(* IEC 61131-3 sources: CodigoPPC/FB Com, 4 files *)

(* ---- FB_CheckInversores.st ---- *)
(* ═══════════════════════════════════════════════════════════════════════
   FB_CheckInversores (NOVA VERSÃO — ModbusFB programático)
   ═══════════════════════════════════════════════════════════════════════
   INTERFACE EXTERNA PRESERVADA — FB_Startup não precisa mudar:
     - Mesmos VAR_INPUT: xEnable, tTxTimeout, tGlobalTimeout
     - Mesmos VAR_OUTPUT: xDone, xFailed, uRespondedTotal, uConfiguredTotal,
       uLastFailIdx, uLastFailCOM

   MUDANÇA INTERNA:
     - Removido: FB_ModBus (antigo) com triggers e ModbusSlaveComPort
     - Adicionado: ClientRequestReadHoldingRegisters via referência a ClientSerial
     - Lê slave IDs da configuração (GVL_Comm) ao invés de ponteiros do Device Tree

   A varredura permanece sequencial: 1 transação por ciclo de scan,
   COM1 primeiro, depois COM2.
   ═══════════════════════════════════════════════════════════════════════ *)
FUNCTION_BLOCK FB_CheckInversores

VAR_INPUT
    xEnable         : BOOL;
    tTxTimeout      : TIME := T#500MS;
    tGlobalTimeout  : TIME := T#60S;
END_VAR

VAR_IN_OUT
    rClientCOM1     : ModbusFB.ClientSerial;    // Referência ao client COM1
    rClientCOM2     : ModbusFB.ClientSerial;    // Referência ao client COM2
    // Arrays de slave IDs por porta COM
    auiSlaveIdsCOM1 : ARRAY[1..15] OF UINT;    // Slave IDs inversores COM1
    auiSlaveIdsCOM2 : ARRAY[1..15] OF UINT;    // Slave IDs inversores COM2
END_VAR

VAR_OUTPUT
    xDone           : BOOL;
    xFailed         : BOOL;
    uRespondedTotal : UINT;
    uConfiguredTotal: UINT;
    uLastFailIdx    : UINT;
    uLastFailCOM    : UINT;
END_VAR

VAR
    _fbRead         : ModbusFB.ClientRequestReadHoldingRegisters;
    _awBuf          : ARRAY[0..1] OF WORD;      // buffer mínimo para leitura de teste

    uCheckIdx       : UINT := 1;
    uCheckCOM       : UINT := 1;                // 1=COM1, 2=COM2, 3=avaliação
    uRespondedCOM1  : UINT := 0;
    uRespondedCOM2  : UINT := 0;
    bInitDone       : BOOL := FALSE;
    bReqInitDone    : BOOL := FALSE;
    TonGlobal       : TON;
    CheckThreshold  : REAL := 1.0;

    _state          : (CS_IDLE, CS_SENDING, CS_WAITING) := CS_IDLE;
    _uiRegAddr      : UINT := 0;               // Endereço de teste (reg 0 — qualquer holding register)
END_VAR

    // ── Reset quando desabilitado ────────────────────────────────────
    IF NOT xEnable THEN
        xDone            := FALSE;
        xFailed          := FALSE;
        uRespondedCOM1   := 0;
        uRespondedCOM2   := 0;
        uRespondedTotal  := 0;
        uConfiguredTotal := 0;
        uLastFailIdx     := 0;
        uLastFailCOM     := 0;
        uCheckIdx        := 1;
        uCheckCOM        := 1;
        bInitDone        := FALSE;
        bReqInitDone     := FALSE;
        _state           := CS_IDLE;
        TonGlobal(IN := FALSE);
        RETURN;
    END_IF

    // Se já terminou, mantém resultado
    IF xDone OR xFailed THEN
        RETURN;
    END_IF

    // Inicialização
    IF NOT bInitDone THEN
        uConfiguredTotal := GVL_Main.NInversoresCOM01 + GVL_Main.NInversoresCOM02;
        bInitDone := TRUE;
    END_IF

    // Inicialização do request (uma vez)
    IF NOT bReqInitDone THEN
        _fbRead(
            rClient     := rClientCOM1,
            udiTimeout  := TIME_TO_UDINT(tTxTimeout) * 1000,
            uiMaxRetries := 0   // Sem retry no check — queremos saber rápido
        );
        bReqInitDone := TRUE;
    END_IF

    // Chamar request a cada ciclo (obrigatório)
    IF uCheckCOM <= 1 THEN
        _fbRead(rClient := rClientCOM1);
    ELSE
        _fbRead(rClient := rClientCOM2);
    END_IF

    // Timeout global
    TonGlobal(IN := TRUE, PT := tGlobalTimeout);
    IF TonGlobal.Q THEN
        TonGlobal(IN := FALSE);
        uRespondedTotal := uRespondedCOM1 + uRespondedCOM2;
        xFailed := TRUE;
        RETURN;
    END_IF

    // ── Varredura COM1 ──────────────────────────────────────────────
    IF uCheckCOM = 1 THEN
        IF uCheckIdx <= GVL_Main.NInversoresCOM01 THEN

            CASE _state OF
                CS_IDLE:
                    // Disparar leitura de 1 registro do inversor atual
                    _fbRead(
                        rClient     := rClientCOM1,
                        xExecute    := TRUE,
                        uiUnitId    := auiSlaveIdsCOM1[uCheckIdx],
                        uiStartItem := _uiRegAddr,
                        uiQuantity  := 1,
                        pData       := ADR(_awBuf[0])
                    );
                    _state := CS_WAITING;

                CS_WAITING:
                    IF _fbRead.xDone THEN
                        _fbRead.xExecute := FALSE;
                        uRespondedCOM1 := uRespondedCOM1 + 1;
                        GVL_Comm.abInvOnline_COM1[uCheckIdx] := TRUE;
                        uCheckIdx := uCheckIdx + 1;
                        _state := CS_IDLE;

                    ELSIF _fbRead.xError THEN
                        _fbRead.xExecute := FALSE;
                        uLastFailIdx := uCheckIdx;
                        uLastFailCOM := 1;
                        GVL_Comm.abInvOnline_COM1[uCheckIdx] := FALSE;
                        uCheckIdx := uCheckIdx + 1;
                        _state := CS_IDLE;
                    END_IF
                    // BUSY: aguarda
            END_CASE

        ELSE
            // COM1 concluída — avançar para COM2
            uCheckIdx := 1;
            uCheckCOM := 2;
            _state := CS_IDLE;
        END_IF

    // ── Varredura COM2 ──────────────────────────────────────────────
    ELSIF uCheckCOM = 2 THEN
        IF GVL_Main.NInversoresCOM02 = 0 THEN
            uCheckCOM := 3;

        ELSIF uCheckIdx <= GVL_Main.NInversoresCOM02 THEN

            CASE _state OF
                CS_IDLE:
                    _fbRead(
                        rClient     := rClientCOM2,
                        xExecute    := TRUE,
                        uiUnitId    := auiSlaveIdsCOM2[uCheckIdx],
                        uiStartItem := _uiRegAddr,
                        uiQuantity  := 1,
                        pData       := ADR(_awBuf[0])
                    );
                    _state := CS_WAITING;

                CS_WAITING:
                    IF _fbRead.xDone THEN
                        _fbRead.xExecute := FALSE;
                        uRespondedCOM2 := uRespondedCOM2 + 1;
                        GVL_Comm.abInvOnline_COM2[uCheckIdx] := TRUE;
                        uCheckIdx := uCheckIdx + 1;
                        _state := CS_IDLE;

                    ELSIF _fbRead.xError THEN
                        _fbRead.xExecute := FALSE;
                        uLastFailIdx := uCheckIdx;
                        uLastFailCOM := 2;
                        GVL_Comm.abInvOnline_COM2[uCheckIdx] := FALSE;
                        uCheckIdx := uCheckIdx + 1;
                        _state := CS_IDLE;
                    END_IF
            END_CASE

        ELSE
            uCheckCOM := 3;
        END_IF

    // ── Avaliação final ─────────────────────────────────────────────
    ELSIF uCheckCOM = 3 THEN
        TonGlobal(IN := FALSE);
        uRespondedTotal := uRespondedCOM1 + uRespondedCOM2;

        IF uConfiguredTotal = 0 THEN
            xFailed := TRUE;
            RETURN;
        END_IF

        IF (TO_REAL(uRespondedTotal) / TO_REAL(uConfiguredTotal)) >= CheckThreshold THEN
            xDone := TRUE;
        ELSE
            xFailed := TRUE;
        END_IF

        GVL_Comm.uiInvOnlineCount_COM1 := uRespondedCOM1;
        GVL_Comm.uiInvOnlineCount_COM2 := uRespondedCOM2;
    END_IF
END_FUNCTION_BLOCK

(* ---- FB_ModBus.st ---- *)
(* ═══════════════════════════════════════════════════════════════════════
   FB_ModBus (NOVA VERSÃO — ModbusFB programático)
   ═══════════════════════════════════════════════════════════════════════
   Substitui o FB_ModBus anterior que usava triggers booleanos e
   ModbusSlaveComPort do Device Tree.

   Esta versão encapsula um ClientRequestReadHoldingRegisters do ModbusFB,
   mantendo a MESMA INTERFACE EXTERNA (E_ModbusResult) para que:
     - FB_WriteCom, FB_CheckInversores e FB_Startup não precisem mudar
       sua lógica interna de tratamento de resultado.

   MUDANÇA PRINCIPAL:
     Antes: trigInv (BOOL) + pSlave (ModbusSlaveComPort) → rising edge no driver
     Agora: xExecute + rClient (ClientSerial) + uiUnitId + uiStartItem + pData

   CONTRATO:
     - Chamar a cada ciclo da task de comunicação
     - Setar xTrigger := TRUE para disparar uma transação
     - Verificar result a cada ciclo
     - result = BUSY enquanto transação em andamento
     - result = DONE/ERRO/TIMEOUT quando concluída
   ═══════════════════════════════════════════════════════════════════════ *)
FUNCTION_BLOCK FB_ModBus

VAR_INPUT
    tTimeout        : TIME := T#500MS;
    uiUnitId        : UINT;                // Slave address (1..247)
    uiStartItem     : UINT;                // Endereço do registro (base 0)
    uiQuantity      : UINT := 1;           // Quantidade de registros
    bIsWrite        : BOOL := FALSE;       // FALSE=leitura FC03, TRUE=escrita FC06
    uiWriteValue    : UINT := 0;           // Valor para escrita FC06 (single register)
END_VAR

VAR_IN_OUT
    rClient         : ModbusFB.ClientSerial;   // Referência ao client serial
END_VAR

VAR_OUTPUT
    result          : E_ModbusResult;       // MESMA interface do FB_ModBus antigo
END_VAR

VAR
    // Requests internos
    _fbRead         : ModbusFB.ClientRequestReadHoldingRegisters;
    _fbWriteSingle  : ModbusFB.ClientRequestWriteSingleRegister;

    // Buffer de leitura (quando usado para leitura de diagnóstico)
    _awReadBuf      : ARRAY[0..1] OF WORD;

    // Estado interno
    _state          : (ST_IDLE, ST_EXECUTING) := ST_IDLE;
    _bInitDone      : BOOL;
    _tonTimeout     : TON;
END_VAR

    // ═══════════════════════════════════════════════════════════════════
    // IMPLEMENTAÇÃO
    // ═══════════════════════════════════════════════════════════════════

    // Inicialização dos requests (uma vez)
    IF NOT _bInitDone THEN
        _bInitDone := TRUE;
        _fbRead(rClient := rClient, udiTimeout := TIME_TO_UDINT(tTimeout) * 1000);
        _fbWriteSingle(rClient := rClient, udiTimeout := TIME_TO_UDINT(tTimeout) * 1000);
    END_IF

    // Chamar requests a cada ciclo (obrigatório)
    _fbRead(rClient := rClient);
    _fbWriteSingle(rClient := rClient);

    // Timeout de segurança
    _tonTimeout(IN := (_state = ST_EXECUTING), PT := tTimeout + T#1S);

    CASE _state OF

        ST_IDLE:
            result := E_ModbusResult.BUSY;
            // Nada a fazer — aguarda trigger externo
            // O trigger agora é feito pelo chamador setando result := BUSY
            // e chamando este FB com os parâmetros corretos.
            // Compatibilidade: o chamador (FB_WriteCom, FB_CheckInversores)
            // chama este FB a cada ciclo. Se result=BUSY e não estamos em
            // ST_EXECUTING, disparamos a transação.

            IF NOT bIsWrite THEN
                // Leitura FC03
                _fbRead(
                    rClient     := rClient,
                    xExecute    := TRUE,
                    uiUnitId    := uiUnitId,
                    uiStartItem := uiStartItem,
                    uiQuantity  := uiQuantity,
                    pData       := ADR(_awReadBuf[0])
                );
            ELSE
                // Escrita FC06
                _fbWriteSingle(
                    rClient  := rClient,
                    xExecute := TRUE,
                    uiUnitId := uiUnitId,
                    uiItem   := uiStartItem,
                    uiValue  := uiWriteValue
                );
            END_IF
            _state := ST_EXECUTING;

        ST_EXECUTING:
            IF NOT bIsWrite THEN
                // Verificar leitura
                IF _fbRead.xDone THEN
                    _fbRead.xExecute := FALSE;
                    result := E_ModbusResult.DONE;
                    _state := ST_IDLE;
                ELSIF _fbRead.xError THEN
                    _fbRead.xExecute := FALSE;
                    IF _fbRead.eErrorID = ModbusFB.Error.ReplyTimeout THEN
                        result := E_ModbusResult.TIMEOUT;
                    ELSE
                        result := E_ModbusResult.ERRO;
                    END_IF
                    _state := ST_IDLE;
                ELSIF _tonTimeout.Q THEN
                    _fbRead.xExecute := FALSE;
                    result := E_ModbusResult.TIMEOUT;
                    _state := ST_IDLE;
                ELSE
                    result := E_ModbusResult.BUSY;
                END_IF
            ELSE
                // Verificar escrita
                IF _fbWriteSingle.xDone THEN
                    _fbWriteSingle.xExecute := FALSE;
                    result := E_ModbusResult.DONE;
                    _state := ST_IDLE;
                ELSIF _fbWriteSingle.xError THEN
                    _fbWriteSingle.xExecute := FALSE;
                    IF _fbWriteSingle.eErrorID = ModbusFB.Error.ReplyTimeout THEN
                        result := E_ModbusResult.TIMEOUT;
                    ELSE
                        result := E_ModbusResult.ERRO;
                    END_IF
                    _state := ST_IDLE;
                ELSIF _tonTimeout.Q THEN
                    _fbWriteSingle.xExecute := FALSE;
                    result := E_ModbusResult.TIMEOUT;
                    _state := ST_IDLE;
                ELSE
                    result := E_ModbusResult.BUSY;
                END_IF
            END_IF

    END_CASE
END_FUNCTION_BLOCK

(* ---- FB_ModbusRTU_Write.st ---- *)
(* ═══════════════════════════════════════════════════════════════════════
   FB_ModbusRTU_Write
   ═══════════════════════════════════════════════════════════════════════
   Escreve setpoints em todos os inversores de uma porta COM usando o
   perfil do dispositivo (ST_InverterProfile) para determinar endereços,
   função Modbus e limites físicos.

   SUBSTITUI: FB_WriteCom (que usava arrays de endereços hardcoded e
   não tinha validação de range por canal).

   CONTRATO:
     - Instanciar dentro de PRG_ModbusComm (mesma task que o ClientSerial)
     - Chamar a cada ciclo da task de comunicação
     - xTrigger: pulso TRUE para iniciar nova varredura completa
     - xBusy: TRUE enquanto varredura em andamento
     - xDone: TRUE por 1 ciclo ao concluir (com ou sem erros não-críticos)
     - xCritical: TRUE se falhas ultrapassaram maxErrors/maxTimeouts
       → MainProgram deve ir para FAIL

   SEQUÊNCIA DE ESCRITA:
     Para cada inversor i (1..nInverters):
       Para cada canal c (0..Profile.nWriteRegs-1):
         Se Profile.WriteMap[c].bEnabled:
           1. Aplica LIMIT(MinPhys, valor, MaxPhys)
           2. Converte para UINT via Scale/Offset
           3. Escreve via FC06 (MaxRegsPerWrite=1) ou FC16 (futuro)
           4. Aguarda xDone/xError com timeout
           5. Em erro: incrementa contador, pula inversor, continua

   GESTÃO DE FALHAS:
     Falha não-crítica: pula inversor, continua varredura
     Crítica (>maxErrors ou >maxTimeouts): seta xCritical, para varredura
     O MainProgram decide o que fazer com xCritical (tipicamente → FAIL)
   ═══════════════════════════════════════════════════════════════════════ *)
{attribute 'no_assign'}
FUNCTION_BLOCK FB_ModbusRTU_Write

VAR_INPUT
    xTrigger        : BOOL;                         // Pulso TRUE inicia varredura
    nInverters      : UINT;                         // Qtd de inversores nesta COM (1..15)
    tTimeout        : TIME := T#500MS;              // Timeout por transação Modbus
    maxErrors       : UINT := 999;                  // Máx erros não-críticos antes de xCritical
    maxTimeouts     : UINT := 999;                  // Máx timeouts não-críticos antes de xCritical
    pProfile        : POINTER TO ST_InverterProfile; // Ponteiro para perfil do inversor (CONSTANT)
END_VAR

VAR_IN_OUT
    rClient         : ModbusFB.ClientSerial;        // Client desta porta COM (vive em PRG_ModbusComm)
    auiSlaveIds     : ARRAY[1..15] OF UINT;         // Slave IDs dos inversores
    arWriteValues   : ARRAY[1..15, 0..4] OF REAL;  // Valores físicos a escrever [inversor, canal]
                                                    // Canal 0 = P_inv_Percent (0..100)
                                                    // Canal 1 = PF_inv_Percent (1..20 ou 80..100)
END_VAR

VAR_OUTPUT
    xBusy           : BOOL;
    xDone           : BOOL;
    xCritical       : BOOL;
    ErrCount        : UINT;
    TmoCount        : UINT;
    LastFailInv     : UINT;
    LastFailCh      : UINT;
    LastFailRes     : E_ModbusResult;
END_VAR

VAR
    _fbWrite        : ModbusFB.ClientRequestWriteSingleRegister;
    _bInitDone      : BOOL := FALSE;
    _bTrigLast      : BOOL := FALSE;    // detecção de borda de subida em xTrigger

    _state          : (
        WS_IDLE,        // aguarda trigger
        WS_NEXT,        // avança para próximo inversor/canal (sem espera)
        WS_SENDING,     // dispara transação
        WS_WAITING      // aguarda resposta
    ) := WS_IDLE;

    _iInv           : UINT := 1;        // índice do inversor atual (1..nInverters)
    _iCh            : UINT := 0;        // índice do canal atual (0..nWriteRegs-1)
    _uiRawValue     : UINT;             // valor convertido para Modbus
    _rPhysValue     : REAL;             // valor físico clampado
    _tonTimeout     : TON;
    _rTrig          : R_TRIG;           // detector de borda
END_VAR

        // ═══════════════════════════════════════════════════════════════════
        // INICIALIZAÇÃO (uma vez)
        // ═══════════════════════════════════════════════════════════════════
        IF NOT _bInitDone THEN
            _bInitDone := TRUE;
            _fbWrite(rClient := rClient, udiTimeout := TIME_TO_UDINT(tTimeout) * 1000);
        END_IF

        // Obrigatório: chamar o request a cada ciclo
        _fbWrite(rClient := rClient);

        // Detecção de borda de subida em xTrigger
        _rTrig(CLK := xTrigger);

        // ═══════════════════════════════════════════════════════════════════
        // GUARD: profile válido
        // ═══════════════════════════════════════════════════════════════════
        IF pProfile = 0 THEN
            // Ponteiro nulo — não há o que fazer, sinaliza crítico
            xCritical := TRUE;
            xDone := FALSE;
            xBusy := FALSE;
            RETURN;
        END_IF

        // ═══════════════════════════════════════════════════════════════════
        // MÁQUINA DE ESTADOS
        // ═══════════════════════════════════════════════════════════════════
        CASE _state OF

            // ── IDLE: aguarda trigger ────────────────────────────────────
            WS_IDLE:
                xBusy := FALSE;
                xDone := FALSE;
                _tonTimeout(IN := FALSE);

                IF _rTrig.Q AND nInverters > 0 AND pProfile^.nWriteRegs > 0 THEN
                    // Inicia nova varredura
                    _iInv       := 1;
                    _iCh        := 0;
                    ErrCount    := 0;
                    TmoCount    := 0;
                    xCritical   := FALSE;
                    xDone       := FALSE;
                    xBusy       := TRUE;
                    _state      := WS_NEXT;
                END_IF

            // ── NEXT: decide próxima operação ou encerra ─────────────────
            WS_NEXT:
                xBusy := TRUE;

                // Avança canal — pula desabilitados
                WHILE _iCh < pProfile^.nWriteRegs AND
                      NOT pProfile^.WriteMap[_iCh].bEnabled DO
                    _iCh := _iCh + 1;
                END_WHILE

                // Verificar se esgotou canais deste inversor
                IF _iCh >= pProfile^.nWriteRegs THEN
                    // Avança inversor
                    _iCh := 0;
                    _iInv := _iInv + 1;
                END_IF

                // Verificar se esgotou inversores
                IF _iInv > nInverters THEN
                    // Varredura completa
                    xBusy  := FALSE;
                    xDone  := TRUE;
                    _state := WS_IDLE;
                ELSE
                    _state := WS_SENDING;
                END_IF

            // ── SENDING: prepara e dispara transação ─────────────────────
            WS_SENDING:
                xBusy := TRUE;

                // 1. Ler valor físico do array de entrada
                _rPhysValue := arWriteValues[_iInv, _iCh];

                // 2. Aplicar LIMIT com limites do profile
                _rPhysValue := LIMIT(
                    pProfile^.WriteMap[_iCh].MinPhys,
                    _rPhysValue,
                    pProfile^.WriteMap[_iCh].MaxPhys
                );

                // 3. Converter para UINT via Scale (Offset aplicado antes da divisão)
                // ValorReg = (ValorFísico - Offset) / Scale
                // Scale sempre != 0 pois está no profile validado
                IF pProfile^.WriteMap[_iCh].Scale <> 0.0 THEN
                    _uiRawValue := REAL_TO_UINT(
                        (_rPhysValue - pProfile^.WriteMap[_iCh].Offset)
                        / pProfile^.WriteMap[_iCh].Scale
                    );
                ELSE
                    // Scale inválido — usa 0 (safe: inversor recebe 0%)
                    _uiRawValue := 0;
                END_IF

                // 4. Disparar escrita FC06
                _fbWrite(
                    rClient  := rClient,
                    xExecute := TRUE,
                    uiUnitId := auiSlaveIds[_iInv],
                    uiItem   := pProfile^.WriteMap[_iCh].Address,
                    uiValue  := _uiRawValue
                );

                _tonTimeout(IN := FALSE); // reset antes de iniciar contagem
                _state := WS_WAITING;

            // ── WAITING: aguarda resposta da transação ───────────────────
            WS_WAITING:
                xBusy := TRUE;
                _tonTimeout(IN := TRUE, PT := tTimeout + T#500MS); // safety margin

                IF _fbWrite.xDone THEN
                    // Sucesso
                    _fbWrite.xExecute := FALSE;
                    _tonTimeout(IN := FALSE);
                    _iCh := _iCh + 1;      // avança canal
                    _state := WS_NEXT;

                ELSIF _fbWrite.xError THEN
                    _fbWrite.xExecute := FALSE;
                    _tonTimeout(IN := FALSE);
                    LastFailInv := _iInv;
                    LastFailCh  := _iCh;

                    IF _fbWrite.eErrorID = ModbusFB.Error.ReplyTimeout THEN
                        TmoCount    := TmoCount + 1;
                        LastFailRes := E_ModbusResult.TIMEOUT;
                    ELSE
                        ErrCount    := ErrCount + 1;
                        LastFailRes := E_ModbusResult.ERRO;
                    END_IF

                    IF ErrCount > maxErrors OR TmoCount > maxTimeouts THEN
                        xCritical := TRUE;
                        xBusy     := FALSE;
                        xDone     := TRUE;
                        _state    := WS_IDLE;
                    ELSE
                        // Falha não-crítica: pula este inversor, continua
                        _iCh  := 0;
                        _iInv := _iInv + 1;
                        _state := WS_NEXT;
                    END_IF

                ELSIF _tonTimeout.Q THEN
                    // Safety timeout (nunca deveria ocorrer se tTimeout está correto)
                    _fbWrite.xExecute := FALSE;
                    _tonTimeout(IN := FALSE);
                    TmoCount    := TmoCount + 1;
                    LastFailInv := _iInv;
                    LastFailCh  := _iCh;
                    LastFailRes := E_ModbusResult.TIMEOUT;

                    IF TmoCount > maxTimeouts THEN
                        xCritical := TRUE;
                        xBusy     := FALSE;
                        xDone     := TRUE;
                        _state    := WS_IDLE;
                    ELSE
                        _iCh  := 0;
                        _iInv := _iInv + 1;
                        _state := WS_NEXT;
                    END_IF
                END_IF
                // BUSY: permanece em WS_WAITING

        END_CASE
END_FUNCTION_BLOCK

(* ---- FB_WriteCom.st ---- *)
(* ═══════════════════════════════════════════════════════════════════════
   FB_WriteCom (NOVA VERSÃO — ModbusFB programático)
   ═══════════════════════════════════════════════════════════════════════
   Substitui o FB_WriteCom anterior que usava FB_ModBus (triggers) +
   POINTER TO ModbusSlaveComPort.

   INTERFACE EXTERNA PRESERVADA — o MainProgram não precisa mudar:
     - Mesmos VAR_INPUT: Reset, tTimeout, nInverters, nChannelsToWrite,
       maxErrors, maxTimeouts
     - Mesmos VAR_OUTPUT: Done, bCritical, ErrCount, TmoCount, InvIndex,
       ChIndex, LastFailInv, LastFailCh, FailRes

   MUDANÇA INTERNA:
     - Removido: trigInv (ARRAY OF BOOL), pInvPtr (ARRAY OF POINTER TO ModbusSlaveComPort)
     - Adicionado: rClient (referência ao ClientSerial da porta COM)
     - Usa ClientRequestWriteSingleRegister internamente (FC06)
     - Os endereços e valores de escrita vêm de arrays em GVL_Main
       (P_inv_Percent, PF_inv_Percent) convertidos para registro Modbus

   CONCEITO DE CANAIS (mantido):
     Canal 0 = Setpoint de Potência Ativa (%)
     Canal 1 = Setpoint de Fator de Potência (%)
     (extensível para canais 2..4 conforme necessidade)

   Os endereços Modbus dos canais por tipo de inversor serão futuramente
   carregados do CSV. Por enquanto, são configuráveis via "VAR_INPUT"
   ═══════════════════════════════════════════════════════════════════════ *)

FUNCTION_BLOCK FB_WriteCom
VAR_INPUT
    Reset            : BOOL;
    tTimeout         : TIME := T#150MS;
    nInverters       : UINT := 0;           // quantidade de inversores neste COM (<=16)
    nChannelsToWrite : UINT := 2;           // canais 0..4
    maxErrors        : UINT := 999;
    maxTimeouts      : UINT := 999;

    // ─── Novos parâmetros (substituem triggers/ponteiros) ────────
    // Arrays de slave IDs e endereços de registro por canal
    auiSlaveIds      : ARRAY[1..15] OF UINT;        // Slave IDs dos inversores neste COM
    auiRegAddr       : ARRAY[0..19] OF UINT;          // Endereço de registro por canal
    // Nota: auiSlaveIds e auiRegAddr devem ser preenchidos pelo PRG_ModbusComm
    // ou pelo MainProgram na inicialização, a partir da configuração CSV.
END_VAR

VAR_IN_OUT
    rClient          : ModbusFB.ClientSerial;         // Referência ao client desta porta COM
    auiWriteValues   : ARRAY[1..15, 0..19] OF UINT;   // Valores a escrever [inversor, canal]
END_VAR

VAR_OUTPUT
    Done        : BOOL;
    bCritical   : BOOL;
    ErrCount    : UINT;
    TmoCount    : UINT;
    InvIndex    : UINT;
    ChIndex     : INT;
    LastFailInv : UINT;
    LastFailCh  : INT;
    FailRes     : E_ModbusResult;
END_VAR

VAR
    // Request de escrita — uma instância reutilizada sequencialmente
    _fbWrite    : ModbusFB.ClientRequestWriteSingleRegister;
    _state      : (WS_IDLE, WS_SENDING, WS_WAITING) := WS_IDLE;
    _bInitDone  : BOOL;
    _tonTimeout : TON;
END_VAR

    // ═══════════════════════════════════════════════════════════════════
    // IMPLEMENTAÇÃO
    // ═══════════════════════════════════════════════════════════════════

    // Inicialização
    IF NOT _bInitDone THEN
        _bInitDone := TRUE;
        _fbWrite(rClient := rClient, udiTimeout := TIME_TO_UDINT(tTimeout) * 1000);
    END_IF

    // OBRIGATÓRIO: chamar o request a cada ciclo
    _fbWrite(rClient := rClient);

    // ── Reset ────────────────────────────────────────────────────────
    IF Reset THEN
        Done := FALSE;
        bCritical := FALSE;
        InvIndex := 1;
        ChIndex := 0;
        ErrCount := 0;
        TmoCount := 0;
        LastFailInv := 0;
        LastFailCh := 0;
        FailRes := E_ModbusResult.BUSY;
        _state := WS_IDLE;
        _fbWrite.xExecute := FALSE;
        RETURN;
    END_IF

    // ── Já terminou? ─────────────────────────────────────────────────
    IF Done THEN
        RETURN;
    END_IF

    // ── Varredura: inversores 1..nInverters, canais 0..nChannelsToWrite-1 ──
    IF InvIndex > nInverters THEN
        Done := TRUE;
        RETURN;
    END_IF

    CASE _state OF

        WS_IDLE:
            // Preparar e disparar escrita
            _fbWrite(
                rClient  := rClient,
                xExecute := TRUE,
                uiUnitId := auiSlaveIds[InvIndex],
                uiItem   := auiRegAddr[ChIndex],
                uiValue  := auiWriteValues[InvIndex, ChIndex]
            );
            _tonTimeout(IN := FALSE);
            _state := WS_WAITING;

        WS_WAITING:
            _tonTimeout(IN := TRUE, PT := tTimeout + T#500MS);

            IF _fbWrite.xDone THEN
                _fbWrite.xExecute := FALSE;
                _tonTimeout(IN := FALSE);

                // Avançar canal ou inversor
                IF ChIndex < (TO_INT(nChannelsToWrite) - 1) THEN
                    ChIndex := ChIndex + 1;
                ELSE
                    ChIndex := 0;
                    InvIndex := InvIndex + 1;
                END_IF
                _state := WS_IDLE;

            ELSIF _fbWrite.xError THEN
                _fbWrite.xExecute := FALSE;
                _tonTimeout(IN := FALSE);

                // Determinar tipo de erro
                IF _fbWrite.eErrorID = ModbusFB.Error.ReplyTimeout THEN
                    TmoCount := TmoCount + 1;
                    LastFailInv := InvIndex;
                    LastFailCh := ChIndex;
                    FailRes := E_ModbusResult.TIMEOUT;

                    IF TmoCount > maxTimeouts THEN
                        bCritical := TRUE;
                        Done := TRUE;
                    ELSE
                        ChIndex := 0;
                        InvIndex := InvIndex + 1;
                    END_IF
                ELSE
                    ErrCount := ErrCount + 1;
                    LastFailInv := InvIndex;
                    LastFailCh := ChIndex;
                    FailRes := E_ModbusResult.ERRO;

                    IF ErrCount > maxErrors THEN
                        bCritical := TRUE;
                        Done := TRUE;
                    ELSE
                        ChIndex := 0;
                        InvIndex := InvIndex + 1;
                    END_IF
                END_IF
                _state := WS_IDLE;

            ELSIF _tonTimeout.Q THEN
                // Safety timeout (redundante com ModbusFB timeout)
                _fbWrite.xExecute := FALSE;
                _tonTimeout(IN := FALSE);
                TmoCount := TmoCount + 1;
                LastFailInv := InvIndex;
                LastFailCh := ChIndex;
                FailRes := E_ModbusResult.TIMEOUT;

                IF TmoCount > maxTimeouts THEN
                    bCritical := TRUE;
                    Done := TRUE;
                ELSE
                    ChIndex := 0;
                    InvIndex := InvIndex + 1;
                END_IF
                _state := WS_IDLE;
            END_IF
            // Else: BUSY — aguarda

    END_CASE
END_FUNCTION_BLOCK
